FUNCTION_BLOCK NeredaReactor_HMI (* Service Interface Function Block Type *)
  (* Standard: 61499-2 *)
  (* Version 0.0, 6/7/2026, Schneider Electric, template *)
  PACKAGE SE.Nereda;
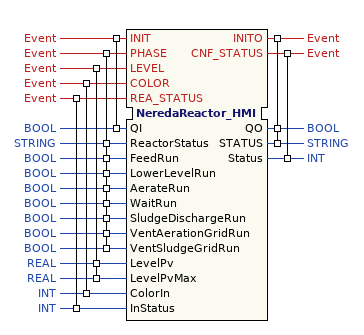
  EVENT_INPUT
    INIT WITH QI;
    PHASE WITH FeedRun, AerateRun, SludgeDischargeRun, VentAerationGridRun, WaitRun, ReactorStatus, VentSludgeGridRun, LowerLevelRun;
    LEVEL WITH LevelPv, LevelPvMax;
    COLOR WITH ColorIn;
    REA_STATUS WITH InStatus;
  END_EVENT
  EVENT_OUTPUT
    INITO WITH QO, STATUS;
    CNF_STATUS WITH Status;
  END_EVENT
  VAR_INPUT
    QI : BOOL;
    ReactorStatus : STRING;
    FeedRun : BOOL;
    LowerLevelRun : BOOL;
    AerateRun : BOOL;
    WaitRun : BOOL;
    SludgeDischargeRun : BOOL;
    VentAerationGridRun : BOOL;
    VentSludgeGridRun : BOOL;
    LevelPv : REAL;
    LevelPvMax : REAL;
    ColorIn : INT;
    InStatus : INT;
  END_VAR
  VAR_OUTPUT
    QO : BOOL; (* Event Output Qualifier *)
    STATUS : STRING; (* Service Status *)
    Status : INT;
  END_VAR
  SERVICE /
    SEQUENCE 
    END_SEQUENCE
  END_SERVICE
END_FUNCTION_BLOCK
